PROGRAM BufferTankFiller
VAR
END_VAR

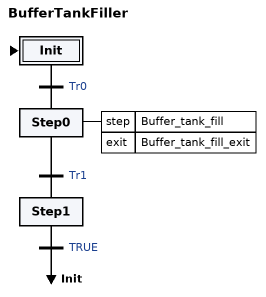
INITIAL_STEP Init:
END_STEP
TRANSITION FROM Init TO Step0
    := Tr0;
END_TRANSITION
STEP Step0:
    Buffer_tank_fill(N);  // step action
    Buffer_tank_fill_exit(P0);  // exit action
END_STEP
TRANSITION FROM Step0 TO Step1
    := Tr1;
END_TRANSITION
STEP Step1:
END_STEP
TRANSITION FROM Step1 TO Init
    := TRUE;
END_TRANSITION

ACTION Buffer_tank_fill:
IF main.LT1mm > 135 THEN
	main.Motor_ON_OFF := FALSE;
ELSIF main.LT1mm < 45 THEN
	main.Motor_ON_OFF := TRUE; 
END_IF
END_ACTION

ACTION Buffer_tank_fill_exit:
main.Motor_ON_OFF := FALSE;
END_ACTION

TRANSITION Tr0:
main.StartBuffer = TRUE;
END_TRANSITION

TRANSITION Tr1:
main.StartBuffer = FALSE;
END_TRANSITION

END_PROGRAM

(* stored: Version 1.1.0.1, ProductVersion 3.1.4024.12
   POU BufferTankFiller: Id {c443e9a3-c137-4c0e-9a28-8b262cd57d43}, SpecialFunc None
   Action Buffer_tank_fill: Id {c167cb7a-6381-4a49-923f-cf5a21c5d22d}
   Action Buffer_tank_fill_exit: Id {63d96bdb-6ec7-4a14-817d-43531ac6a7fc}
   Transition Tr0: Id {4bd19a47-ab37-4114-aeb4-44c0d84ba2f8}
   Transition Tr1: Id {cf1a76e1-0826-4b64-9e49-4efcb26443aa} *)
